{attribute 'qualified_only'}
//{attribute 'strict'}
{attribute 'to_string'}

TYPE E_Util_State_Cmd :
(
	Idle		:= 0,
	Warmup 		:= 1,
	Activate 	:= 2,
	Shutdown 	:= 3,
	Reset_Fault := 4
);
END_TYPE

(* stored: Version 1.1.0.1, ProductVersion 3.1.4024.12
   DUT E_Util_State_Cmd: Id {df7a1b8c-e0e9-43aa-bb32-e2425cb4fe25} *)
